// TwinCAT 3 PLC project PLC1
// ProgramVersion: 3.1.4024.0
// libraries:
//   Tc2_Standard, * (Beckhoff Automation GmbH)
//   Tc2_System, * (Beckhoff Automation GmbH)
//   Tc3_Module, * (Beckhoff Automation GmbH)
// project tree:
//   DUTs/ TestFub.TcPOU, ITestInterface.TcIO, TestFubI.TcPOU, TestStructure.TcDUT
//   GVLs/ GVL.TcGVL
//   / PlcTask.TcTTO
//   POUs/ MAIN.TcPOU
// real-time tasks:
//   TASK PlcTask: cycle T#10ms, priority 20, ADS port 350

CONFIGURATION PLC1
    RESOURCE PLC ON TwinCAT3
        TASK PlcTask(INTERVAL := T#10ms, PRIORITY := 20);
        PROGRAM MAIN WITH PlcTask : MAIN;
    END_RESOURCE
END_CONFIGURATION

// ---- DUTs/TestStructure.TcDUT
TYPE TestStructure :
STRUCT	
	_bool: BOOL;
	_BYTE: BYTE;
	_DATE: DATE;
	_DATE_AND_TIME: DATE_AND_TIME;
	_DINT: DINT;
	_DT: DT;
	_DWORD: DWORD;
	_INT: INT;
	_LINT: LINT;
	_LREAL: LREAL;
	_LTIME: LTIME;
	_LWORD: LWORD;
	_REAL: REAL;
	_SINT: SINT;
	_STRING: STRING;
	_TIME: TIME;
	_TIME_OF_DAY: TIME_OF_DAY;
	_TOD: TOD;
	_UDINT: UDINT;
	_UINT: UINT;
	_ULINT: ULINT;	
	_USINT: USINT;	
	_WORD: WORD;	
	_WSTRING: WSTRING;		
END_STRUCT
END_TYPE

// ---- GVLs/GVL.TcGVL
{attribute 'qualified_only'}
VAR_GLOBAL
	MyFub : TestFub;
	MyStruct: TestStructure; 	
END_VAR

// ---- DUTs/ITestInterface.TcIO
INTERFACE ITestInterface

{attribute 'monitoring' := 'call'}
PROPERTY TestPropGet : BOOL
GET
END_GET
END_PROPERTY

{attribute 'monitoring' := 'call'}
PROPERTY TestPropGetSet : BOOL
GET
END_GET
SET
END_SET
END_PROPERTY

PROPERTY TestPropNoMon : BOOL
GET
END_GET
SET
END_SET
END_PROPERTY

{attribute 'monitoring' := 'call'}
PROPERTY TestPropSet : BOOL
SET
END_SET
END_PROPERTY

END_INTERFACE

// ---- POUs/MAIN.TcPOU
PROGRAM MAIN
VAR
	MyFub : TestFub;
	MyFubI : TestFubI;
	MyStruct: TestStructure; 
END_VAR

MyFub._INTERFACE := MyFubI;
MyFub.Incrementing	:= MyFub.Incrementing + 1;

END_PROGRAM

// ---- DUTs/TestFub.TcPOU
FUNCTION_BLOCK TestFub
VAR_INPUT
	_INTERFACE : ITestInterface;	
	Incrementing : UINT;
END_VAR
VAR
	_bool: BOOL;
	_BYTE: BYTE;
	_DATE: DATE;
	_DATE_AND_TIME: DATE_AND_TIME;
	_DINT: DINT;
	_DT: DT;
	_DWORD: DWORD;
	_INT: INT;
	_LINT: LINT;
	_LREAL: LREAL;
	_LTIME: LTIME;
	_LWORD: LWORD;
	_REAL: REAL;
	_SINT: SINT;
	_STRING: STRING;
	_TIME: TIME;
	_TIME_OF_DAY: TIME_OF_DAY;
	_TOD: TOD;
	_UDINT: UDINT;
	_UINT: UINT;
	_ULINT: ULINT;	
	_USINT: USINT;	
	_WORD: WORD;	
	_WSTRING: WSTRING;	
	_REAL_Array: ARRAY[0..4] OF REAL;
	_STRUCT : TestStructure;
	_INTERFACEEmpty : ITestInterface;
END_VAR

METHOD TestMethod : UINT
VAR_INPUT
END_VAR
END_METHOD

{attribute 'monitoring' := 'call'}
PROPERTY TestPropGet : BOOL
GET
TestPropGet := _bool;
END_GET
END_PROPERTY

{attribute 'monitoring' := 'call'}
PROPERTY TestPropGetSet : BOOL
GET
TestPropGetSet := _bool;
END_GET
SET
_bool := TestPropGetSet;
END_SET
END_PROPERTY

PROPERTY TestPropNoMon : BOOL
GET
TestPropNoMon := _bool;
END_GET
SET
_bool := TestPropNoMon;
END_SET
END_PROPERTY

{attribute 'monitoring' := 'call'}
PROPERTY TestPropSet : BOOL
SET
_bool := TestPropSet;
END_SET
END_PROPERTY

END_FUNCTION_BLOCK

// ---- DUTs/TestFubI.TcPOU
FUNCTION_BLOCK TestFubI IMPLEMENTS ITestInterface
VAR_INPUT
END_VAR
VAR_OUTPUT
END_VAR
VAR
END_VAR

{warning 'add property implementation'}
PROPERTY TestPropGet : BOOL
GET
END_GET
END_PROPERTY

{warning 'add property implementation'}
PROPERTY TestPropGetSet : BOOL
GET
END_GET
SET
END_SET
END_PROPERTY

{warning 'add property implementation'}
PROPERTY TestPropNoMon : BOOL
GET
END_GET
SET
END_SET
END_PROPERTY

{warning 'add property implementation'}
PROPERTY TestPropSet : BOOL
SET
END_SET
END_PROPERTY

END_FUNCTION_BLOCK
